# EPICS substitutions: dma4500mSup/dma4500m_error_setter.substitutions
file $(UTILITIES)/db/error_setter.template {
    pattern {P, STREAM_PV, PV_NAME}

    {"\$(P)", ":MEASUREMENT", ":DENSITY"}
    {"\$(P)", ":MEASUREMENT", ":TEMPERATURE"}
    {"\$(P)", ":MEASUREMENT", ":CONDITION"}
}
